FUNCTION_BLOCK fbLVDT
VAR_INPUT
END_VAR
VAR_OUTPUT
END_VAR
VAR
END_VAR

END_FUNCTION_BLOCK

(* stored: Version 1.1.0.1, ProductVersion 3.1.4024.12
   POU fbLVDT: Id {bb059efb-54fb-4fee-9451-10b597ccd0c6}, SpecialFunc None *)
